FUNCTION_BLOCK Example EXTENDS tcunit.FB_TestSuite
VAR_INPUT
END_VAR
VAR_OUTPUT
END_VAR
VAR
	initWHAT				: BOOL			:= TRUE;
	initRetains 			: BOOL 			:= TRUE;
	inCopyCode 				: BOOL 			:= TRUE;
	count 					: INT 			:= 0;
	count2					: INT 			:= 0;
	currentTestNotZero		: POINTER TO FB_TestSuite;
END_VAR

IF initWHAT THEN
	initWHAT := FALSE;
	count := count + 1;
END_IF;
count2 := count2 + 1;

IF 	TcUnit.GVL_TcUnit.CurrentTestSuiteBeingCalled <> 0 THEN
	currentTestNotZero := TcUnit.GVL_TcUnit.CurrentTestSuiteBeingCalled;
END_IF

TcUnit.GVL_TcUnit.CurrentTestSuiteBeingCalled;

exampleFail();
examplePass();

// base test example for fail
METHOD exampleFail
VAR_INPUT
END_VAR
TEST('ExampleTestFail');
IF TcUnit.GVL_TcUnit.CurrentTestSuiteBeingCalled <> 0 THEN
	currentTestNotZero := TcUnit.GVL_TcUnit.CurrentTestSuiteBeingCalled;
END_IF

TcUnit.GVL_TcUnit.CurrentTestSuiteBeingCalled; 
// @TEST-RUN


// @TEST-ASSERT
AssertTrue(Condition := FALSE,
             Message := 'Test Failed Correctly');// $'emergency error code$' failed at $'diagnostic code type$'');


TEST_FINISHED();
END_METHOD

// base test example for pass
METHOD examplePass
VAR_INPUT
END_VAR
TEST('ExampleTestPass');
 
// @TEST-RUN


// @TEST-ASSERT
AssertTrue(Condition := TRUE,
             Message := 'Test should have passed');

 
TEST_FINISHED();
END_METHOD

END_FUNCTION_BLOCK

(* stored: Version 1.1.0.1, ProductVersion 3.1.4024.12
   POU Example: Id {4c307131-a563-4202-9f15-83919d97ee16}, SpecialFunc None
   Method exampleFail: Id {149bc7a0-64a6-4f67-80d2-60b56815ec6a}
   Method examplePass: Id {58f1b5b4-f723-40ad-ac85-13574514721b} *)
